{attribute 'GeneratedUsingTerminal: EL6688-0000-0017'}
{attribute addProperty BoxType "EL6688-0000-0017"}
{attribute addProperty Id "Sync_ModeAT %I*BYTE1Control_value_update_toggleAT %I*BOOL1Time_stamp_update_toggleAT %I*BOOL1External_device_not_connectedAT %I*BOOL1Internal_time_stampAT %I*ULINT8External_time_stampAT %I*ULINT8Control_Value_for_DC_Master_ClockAT %I*DINT4"}
{attribute addProperty CRC "1767071128"}
{attribute addProperty Size "24"}
TYPE External_Sync_69535D98 EXTENDS InputBase_8311D824 :
STRUCT
	{attribute addProperty Name "Sync_Mode"}
	Sync_Mode AT %I* : BYTE;
	{attribute addProperty Name "Control_value_update_toggle"}
	Control_value_update_toggle AT %I* : BOOL;
	{attribute addProperty Name "Time_stamp_update_toggle"}
	Time_stamp_update_toggle AT %I* : BOOL;
	{attribute addProperty Name "External_device_not_connected"}
	External_device_not_connected AT %I* : BOOL;
	{attribute addProperty Name "Internal_time_stamp"}
	Internal_time_stamp AT %I* : ULINT;
	{attribute addProperty Name "External_time_stamp"}
	External_time_stamp AT %I* : ULINT;
	{attribute addProperty Name "Control_Value_for_DC_Master_Clock"}
	Control_Value_for_DC_Master_Clock AT %I* : DINT;
END_STRUCT
END_TYPE

(* stored: Version 1.2.0.0, ProductVersion 3.1.4024.9
   DUT External_Sync_69535D98: Id {f1d1efc6-0cc7-4262-8d63-a57f91bedc03} *)
